(* Logix 5000 project; controller CarbonScout_MK6 vendor 1 type 14 code 154 rev 32.11; software revision 32.00; part 12 of 17 *)
(* tags used below, declared in another part *)
   DN_Cal : BOOL;   // Calculation Done Bit to proceed next step
   ExtraValvesAuto : BOOL;
   Index : DINT;
   InitialPurgeRequired : BOOL;
   LocalSampleTank : DINT;
   ONS : BOOL[32];
   TimeCompare : TimerCompare;
   AI_LIT_01 : P_AIn;   // Carbon Scout Laser Level Transmitter
   AI_LIT_02 : P_AIn;   // Carbon Scout Cone Level Transmitter
   AI_WIT_01 : P_AIn;   // Weight measure
   CS_Alarms : P_Alarm[80];
   CS_DINTParams : DINT[100];
   CS_REALParams : REAL[80];   // CS REAL Parameters
   CS_Result : CS_Results;   // Sample Result Live Async
   CS_ResultStore : CS_Results[20,20];   // Sample Result Historical
   CS_SampleSeq : DINT[129];
   CS_Seq : GEK_Sequence;
   CS_Seq_ControlStop : BOOL;
   CS_Tank : CS_TankParams[20];
   CS_TankOrder : DINT[17];
   CS_Timer : TIMER[80];
   CS_XRF : XRF;
   CS_XRF_DetTemp : REAL;   // Used in ewon for data records
   CS_XRF_ProbeTemp : REAL;
   FOQ01 : TOTALIZER;   // PurgeTotaliser
   N51 : DINT[5];   // From Client
   Oneshot2 : DINT;
   Oneshot3 : DINT;
   Simulation : DINT;
   TankPointer : DINT;
   TimeAndDate : DINT[7];
   Valve_SPR_01 : P_ValveSO;   // Air injection valve
   Valve_XV_01 : P_ValveSO;   // Sample Valve Tank 1
   Valve_XV_02 : P_ValveSO;   // Sample Valve Tank 2
   Valve_XV_03 : P_ValveSO;   // Sample Valve Tank 3
   Valve_XV_04 : P_ValveSO;   // Sample Valve Tank 4
   Valve_XV_05 : P_ValveSO;   // Sample Valve Tank 5
   Valve_XV_06 : P_ValveSO;   // Sample Valve Tank 6
   Valve_XV_07 : P_ValveSO;   // Sample Valve Tank 7
   Valve_XV_08 : P_ValveSO;   // Sample Valve Tank 8
   Valve_XV_09 : P_ValveSO;   // Sample Valve Tank 9
   Valve_XV_10 : P_ValveSO;   // Sample Valve Tank 10
   Valve_XV_11 : P_ValveSO;   // Purge Valve
   Valve_XV_12 : P_ValveSO;   // Slurry inlet vavle
   Valve_XV_13 : P_ValveSO;   // Sample line vavle
   Valve_XV_14 : P_ValveSO;   // Top wash vavle
   Valve_XV_15 : P_ValveSO;   // Bottme wash vavle
   Valve_XV_16 : P_ValveSO;   // Potable water valve / Supply Water Valve
   Valve_XV_17 : P_ValveSO;   // Sample cone outlet vavle
   Valve_XV_18 : P_ValveSO;   // Sample strainer discharge
   Valve_XV_19 : P_ValveSO;   // Laser window
   Valve_XV_21_30 : P_ValveSO;   // Sample isolation valve
   Valve_XV_30 : P_ValveSO;   // XRF cooling valve
   Valve_XV_40 : P_ValveSO;   // XRF power on valve
   XV2130ClosedOnce : BOOL;
(* SeqProgram, continued *)

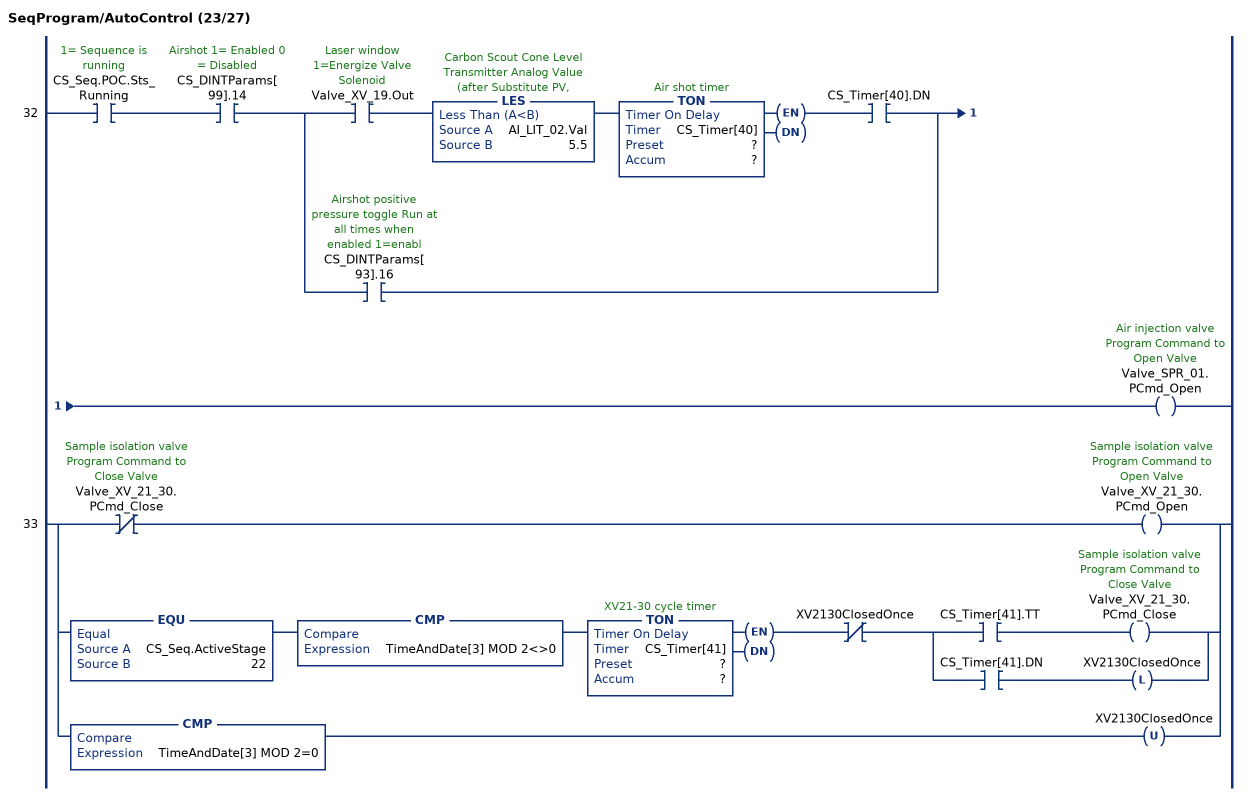
   [picture p234: SeqProgram/AutoControl rungs 32-33]
   32: XIC(CS_Seq.POC.Sts_Running)XIC(CS_DINTParams[99].14)[XIC(Valve_XV_19.Out) LES(AI_LIT_02.Val,5.5) TON(CS_Timer[40],?,?) XIC(CS_Timer[40].DN) ,XIC(CS_DINTParams[93].16) ]OTE(Valve_SPR_01.PCmd_Open);
   33: [XIO(Valve_XV_21_30.PCmd_Close) OTE(Valve_XV_21_30.PCmd_Open) ,EQU(CS_Seq.ActiveStage,22) CMP(TimeAndDate[3] MOD 2<>0) TON(CS_Timer[41],?,?) XIO(XV2130ClosedOnce) [XIC(CS_Timer[41].TT) OTE(Valve_XV_21_30.PCmd_Close) ,XIC(CS_Timer[41].DN) OTL(XV2130ClosedOnce) ] ,CMP(TimeAndDate[3] MOD 2=0) OTU(XV2130ClosedOnce) ];
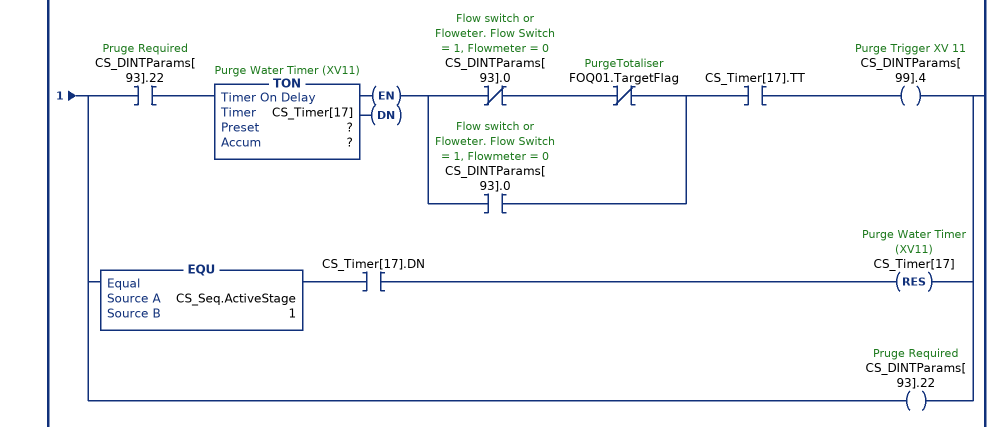
   // Purge Requests
   34: [[[[XIC(CS_DINTParams[99].28) ,XIC(InitialPurgeRequired) ] EQU(CS_Seq.ActiveStage,4) ,EQU(CS_Seq.ActiveStage,13) ] ,XIC(CS_DINTParams[99].4) ] XIC(CS_Seq.POC.Sts_Running) ,[EQU(CS_DINTParams[2],1) XIC(CS_Alarms[14].Alm) XIC(Valve_XV_12.Sts_Closed) ,EQU(CS_DINTParams[2],2) XIC(CS_Alarms[15].Alm) XIC(Valve_XV_12.Sts_Closed) ,EQU(CS_DINTParams[2],3) XIC(CS_Alarms[16].Alm) XIC(Valve_XV_12.Sts_Closed) ,EQU(CS_DINTParams[2],4) XIC(CS_Alarms[17].Alm) XIC(Valve_XV_12.Sts_Closed) ,EQU(CS_DINTParams[2],5) XIC(CS_Alarms[18].Alm) XIC(Valve_XV_12.Sts_Closed) ,EQU(CS_DINTParams[2],6) XIC(CS_Alarms[19].Alm) XIC(Valve_XV_12.Sts_Closed) ,EQU(CS_DINTParams[2],7) XIC(CS_Alarms[20].Alm) XIC(Valve_XV_12.Sts_Closed) ,EQU(CS_DINTParams[2],8) XIC(CS_Alarms[21].Alm) XIC(Valve_XV_12.Sts_Closed) ,EQU(CS_DINTParams[2],9) XIC(CS_Alarms[22].Alm) XIC(Valve_XV_12.Sts_Closed) ,EQU(CS_DINTParams[2],10) XIC(CS_Alarms[23].Alm) XIC(Valve_XV_12.Sts_Closed) ,XIC(CS_DINTParams[99].18) [EQU(CS_DINTParams[2],11) XIC(CS_Alarms[57].Alm) XIC(Valve_XV_12.Sts_Closed) ,EQU(CS_DINTParams[2],12) XIC(CS_Alarms[58].Alm) XIC(Valve_XV_12.Sts_Closed) ,EQU(CS_DINTParams[2],13) XIC(CS_Alarms[59].Alm) XIC(Valve_XV_12.Sts_Closed) ,EQU(CS_DINTParams[2],14) XIC(CS_Alarms[60].Alm) XIC(Valve_XV_12.Sts_Closed) ,EQU(CS_DINTParams[2],15) XIC(CS_Alarms[61].Alm) XIC(Valve_XV_12.Sts_Closed) ,EQU(CS_DINTParams[2],16) XIC(CS_Alarms[62].Alm) XIC(Valve_XV_12.Sts_Closed) ] ] XIO(CS_Seq.POC.Sts_Running) ][XIC(CS_DINTParams[93].22) TON(CS_Timer[17],?,?) [XIO(CS_DINTParams[93].0) XIO(FOQ01.TargetFlag) ,XIC(CS_DINTParams[93].0) ] XIC(CS_Timer[17].TT) OTE(CS_DINTParams[99].4) ,EQU(CS_Seq.ActiveStage,1) XIC(CS_Timer[17].DN) RES(CS_Timer[17]) ,OTE(CS_DINTParams[93].22) ];
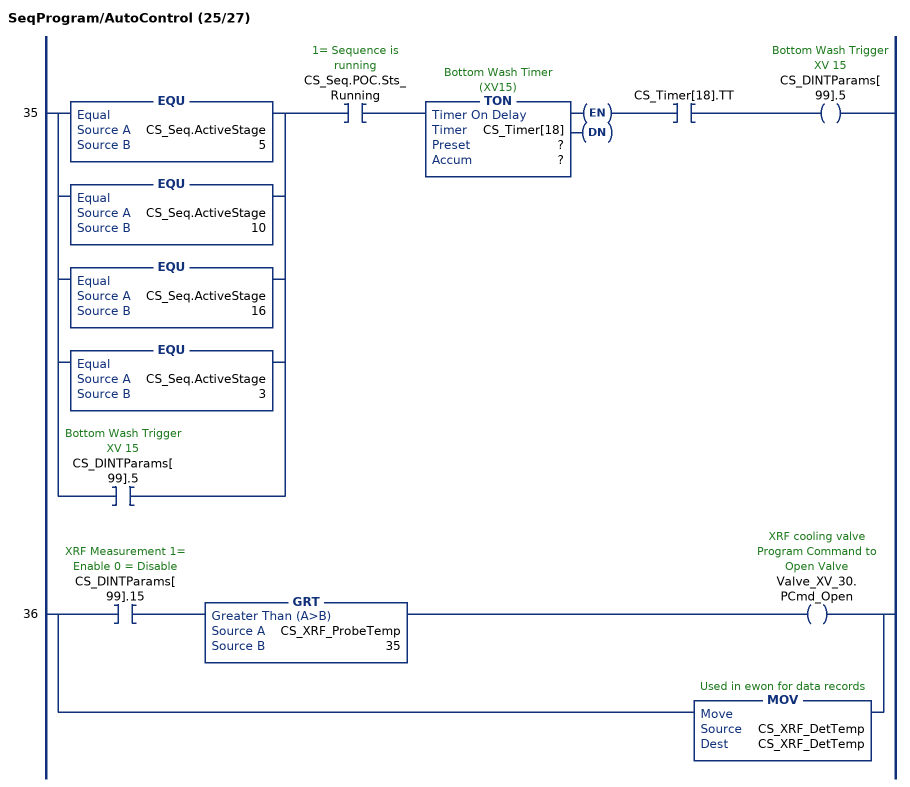
   35: [[EQU(CS_Seq.ActiveStage,5) ,EQU(CS_Seq.ActiveStage,10) ,EQU(CS_Seq.ActiveStage,16) ,EQU(CS_Seq.ActiveStage,3) ] ,XIC(CS_DINTParams[99].5) ]XIC(CS_Seq.POC.Sts_Running)TON(CS_Timer[18],?,?)XIC(CS_Timer[18].TT)OTE(CS_DINTParams[99].5);
   36: [XIC(CS_DINTParams[99].15) GRT(CS_XRF_ProbeTemp,35) OTE(Valve_XV_30.PCmd_Open) ,MOV(CS_XRF_DetTemp,CS_XRF_DetTemp) ];
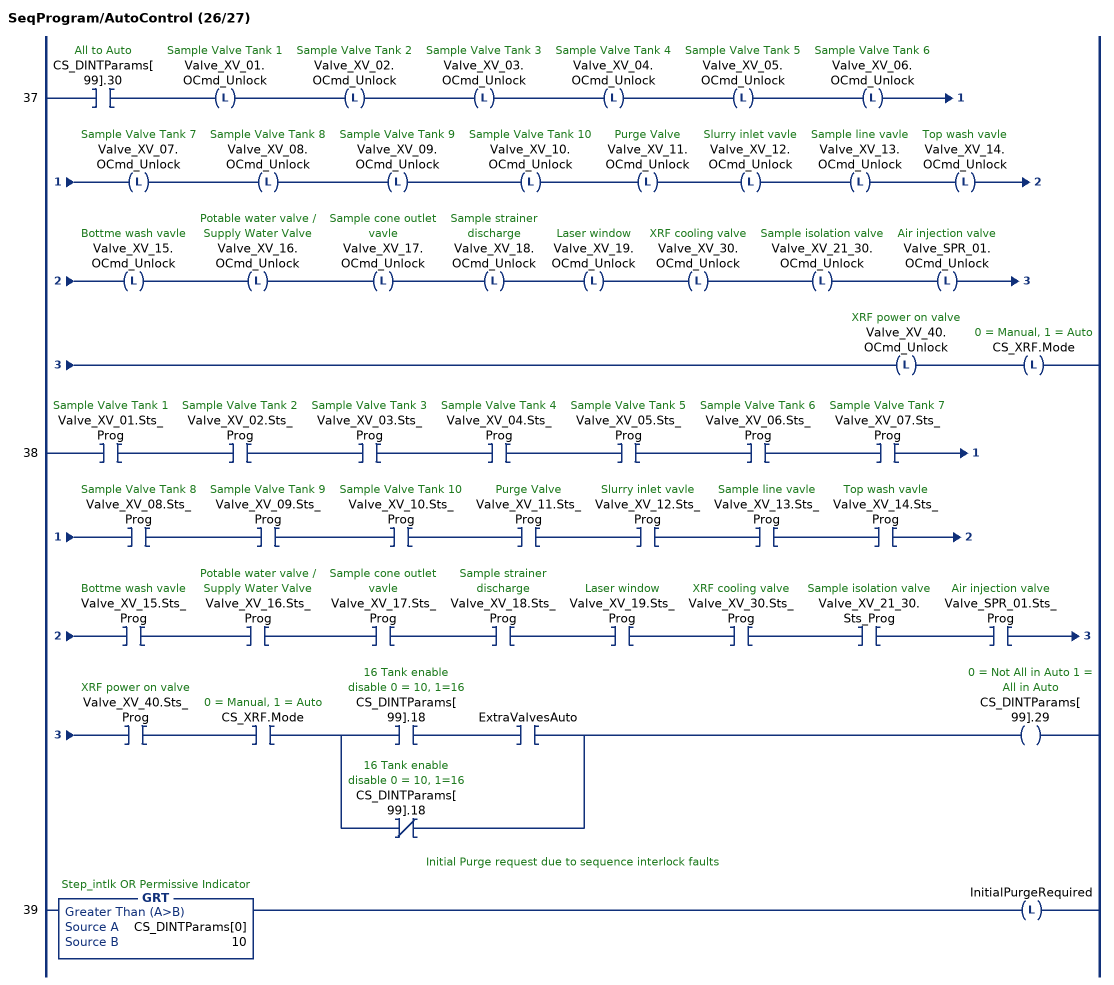
   37: XIC(CS_DINTParams[99].30)OTL(Valve_XV_01.OCmd_Unlock)OTL(Valve_XV_02.OCmd_Unlock)OTL(Valve_XV_03.OCmd_Unlock)OTL(Valve_XV_04.OCmd_Unlock)OTL(Valve_XV_05.OCmd_Unlock)OTL(Valve_XV_06.OCmd_Unlock)OTL(Valve_XV_07.OCmd_Unlock)OTL(Valve_XV_08.OCmd_Unlock)OTL(Valve_XV_09.OCmd_Unlock)OTL(Valve_XV_10.OCmd_Unlock)OTL(Valve_XV_11.OCmd_Unlock)OTL(Valve_XV_12.OCmd_Unlock)OTL(Valve_XV_13.OCmd_Unlock)OTL(Valve_XV_14.OCmd_Unlock)OTL(Valve_XV_15.OCmd_Unlock)OTL(Valve_XV_16.OCmd_Unlock)OTL(Valve_XV_17.OCmd_Unlock)OTL(Valve_XV_18.OCmd_Unlock)OTL(Valve_XV_19.OCmd_Unlock)OTL(Valve_XV_30.OCmd_Unlock)OTL(Valve_XV_21_30.OCmd_Unlock)OTL(Valve_SPR_01.OCmd_Unlock)OTL(Valve_XV_40.OCmd_Unlock)OTL(CS_XRF.Mode);
   38: XIC(Valve_XV_01.Sts_Prog)XIC(Valve_XV_02.Sts_Prog)XIC(Valve_XV_03.Sts_Prog)XIC(Valve_XV_04.Sts_Prog)XIC(Valve_XV_05.Sts_Prog)XIC(Valve_XV_06.Sts_Prog)XIC(Valve_XV_07.Sts_Prog)XIC(Valve_XV_08.Sts_Prog)XIC(Valve_XV_09.Sts_Prog)XIC(Valve_XV_10.Sts_Prog)XIC(Valve_XV_11.Sts_Prog)XIC(Valve_XV_12.Sts_Prog)XIC(Valve_XV_13.Sts_Prog)XIC(Valve_XV_14.Sts_Prog)XIC(Valve_XV_15.Sts_Prog)XIC(Valve_XV_16.Sts_Prog)XIC(Valve_XV_17.Sts_Prog)XIC(Valve_XV_18.Sts_Prog)XIC(Valve_XV_19.Sts_Prog)XIC(Valve_XV_30.Sts_Prog)XIC(Valve_XV_21_30.Sts_Prog)XIC(Valve_SPR_01.Sts_Prog)XIC(Valve_XV_40.Sts_Prog)XIC(CS_XRF.Mode)[XIC(CS_DINTParams[99].18) XIC(ExtraValvesAuto) ,XIO(CS_DINTParams[99].18) ]OTE(CS_DINTParams[99].29);
   // Initial Purge request due to sequence interlock faults
   39: GRT(CS_DINTParams[0],10)OTL(InitialPurgeRequired);
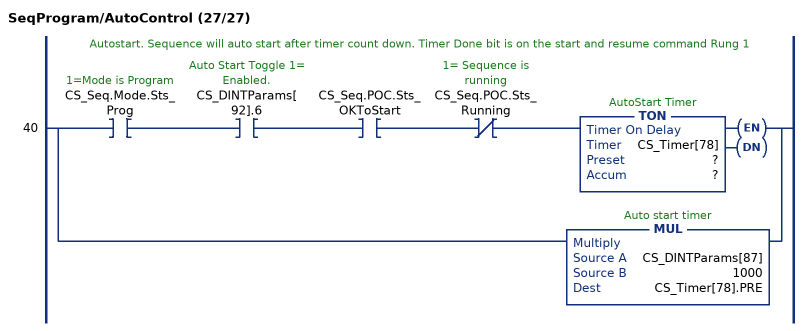
   // Autostart. Sequence will auto start after timer count down. Timer Done bit is on the start and resume command Rung 1
   40: [XIC(CS_Seq.Mode.Sts_Prog) XIC(CS_DINTParams[92].6) XIC(CS_Seq.POC.Sts_OKToStart) XIO(CS_Seq.POC.Sts_Running) TON(CS_Timer[78],?,?) ,MUL(CS_DINTParams[87],1000,CS_Timer[78].PRE) ];
END_ROUTINE

ROUTINE AutoTransition   (* ladder *)
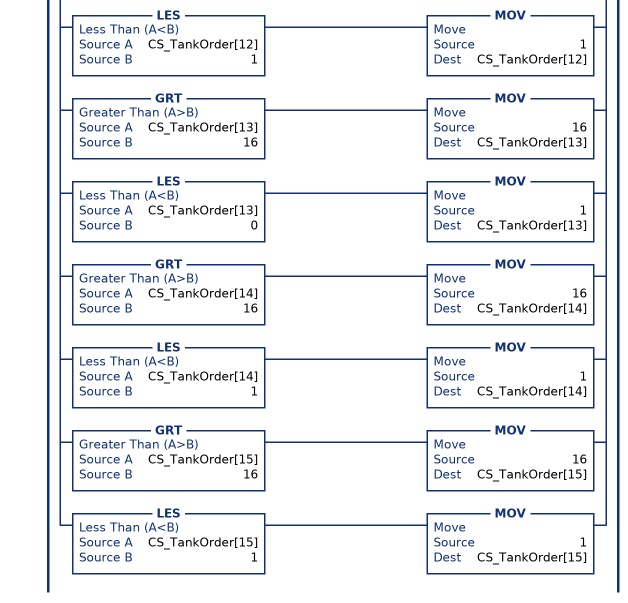
   // Tank order capping
   0: [GRT(CS_TankOrder[0],16) MOV(16,CS_TankOrder[0]) ,LES(CS_TankOrder[0],1) MOV(1,CS_TankOrder[0]) ,GRT(CS_TankOrder[1],16) MOV(16,CS_TankOrder[1]) ,LES(CS_TankOrder[1],1) MOV(1,CS_TankOrder[1]) ,GRT(CS_TankOrder[2],16) MOV(16,CS_TankOrder[2]) ,LES(CS_TankOrder[2],1) MOV(1,CS_TankOrder[2]) ,GRT(CS_TankOrder[3],16) MOV(16,CS_TankOrder[3]) ,LES(CS_TankOrder[3],1) MOV(1,CS_TankOrder[3]) ,GRT(CS_TankOrder[4],16) MOV(16,CS_TankOrder[4]) ,LES(CS_TankOrder[4],1) MOV(1,CS_TankOrder[4]) ,GRT(CS_TankOrder[5],16) MOV(16,CS_TankOrder[5]) ,LES(CS_TankOrder[5],1) MOV(1,CS_TankOrder[5]) ,GRT(CS_TankOrder[6],16) MOV(16,CS_TankOrder[6]) ,LES(CS_TankOrder[6],1) MOV(1,CS_TankOrder[6]) ,GRT(CS_TankOrder[7],16) MOV(16,CS_TankOrder[7]) ,LES(CS_TankOrder[7],1) MOV(1,CS_TankOrder[7]) ,GRT(CS_TankOrder[8],16) MOV(16,CS_TankOrder[8]) ,LES(CS_TankOrder[8],1) MOV(1,CS_TankOrder[8]) ,GRT(CS_TankOrder[9],16) MOV(16,CS_TankOrder[9]) ,LES(CS_TankOrder[9],1) MOV(1,CS_TankOrder[9]) ,GRT(CS_TankOrder[10],16) MOV(16,CS_TankOrder[10]) ,LES(CS_TankOrder[10],1) MOV(1,CS_TankOrder[10]) ,GRT(CS_TankOrder[11],16) MOV(16,CS_TankOrder[11]) ,LES(CS_TankOrder[11],1) MOV(1,CS_TankOrder[11]) ,GRT(CS_TankOrder[12],16) MOV(16,CS_TankOrder[12]) ,LES(CS_TankOrder[12],1) MOV(1,CS_TankOrder[12]) ,GRT(CS_TankOrder[13],16) MOV(16,CS_TankOrder[13]) ,LES(CS_TankOrder[13],0) MOV(1,CS_TankOrder[13]) ,GRT(CS_TankOrder[14],16) MOV(16,CS_TankOrder[14]) ,LES(CS_TankOrder[14],1) MOV(1,CS_TankOrder[14]) ,GRT(CS_TankOrder[15],16) MOV(16,CS_TankOrder[15]) ,LES(CS_TankOrder[15],1) MOV(1,CS_TankOrder[15]) ];
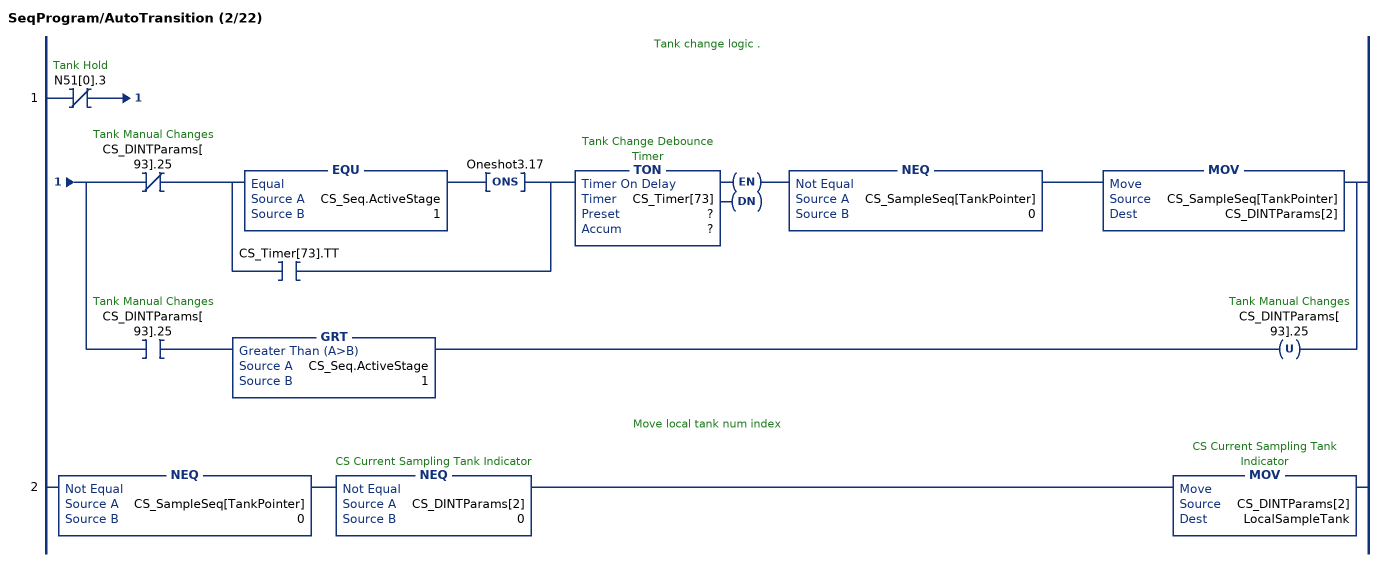
   // Tank change logic .
   1: XIO(N51[0].3)[XIO(CS_DINTParams[93].25) [EQU(CS_Seq.ActiveStage,1) ONS(Oneshot3.17) ,XIC(CS_Timer[73].TT) ] TON(CS_Timer[73],?,?) NEQ(CS_SampleSeq[TankPointer],0) MOV(CS_SampleSeq[TankPointer],CS_DINTParams[2]) ,XIC(CS_DINTParams[93].25) GRT(CS_Seq.ActiveStage,1) OTU(CS_DINTParams[93].25) ];
   // Move local tank num index
   2: NEQ(CS_SampleSeq[TankPointer],0)NEQ(CS_DINTParams[2],0)MOV(CS_DINTParams[2],LocalSampleTank);
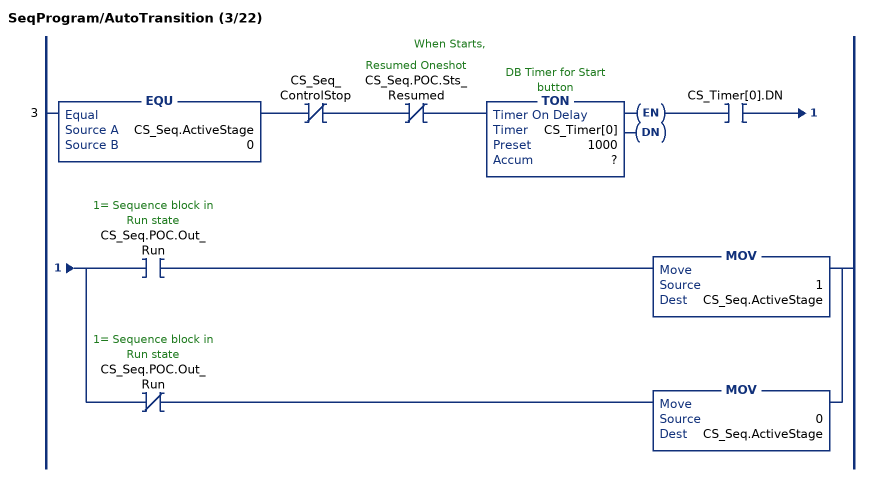
   // When Starts,
   3: EQU(CS_Seq.ActiveStage,0)XIO(CS_Seq_ControlStop)XIO(CS_Seq.POC.Sts_Resumed)TON(CS_Timer[0],?,?)XIC(CS_Timer[0].DN)[XIC(CS_Seq.POC.Out_Run) MOV(1,CS_Seq.ActiveStage) ,XIO(CS_Seq.POC.Out_Run) MOV(0,CS_Seq.ActiveStage) ];
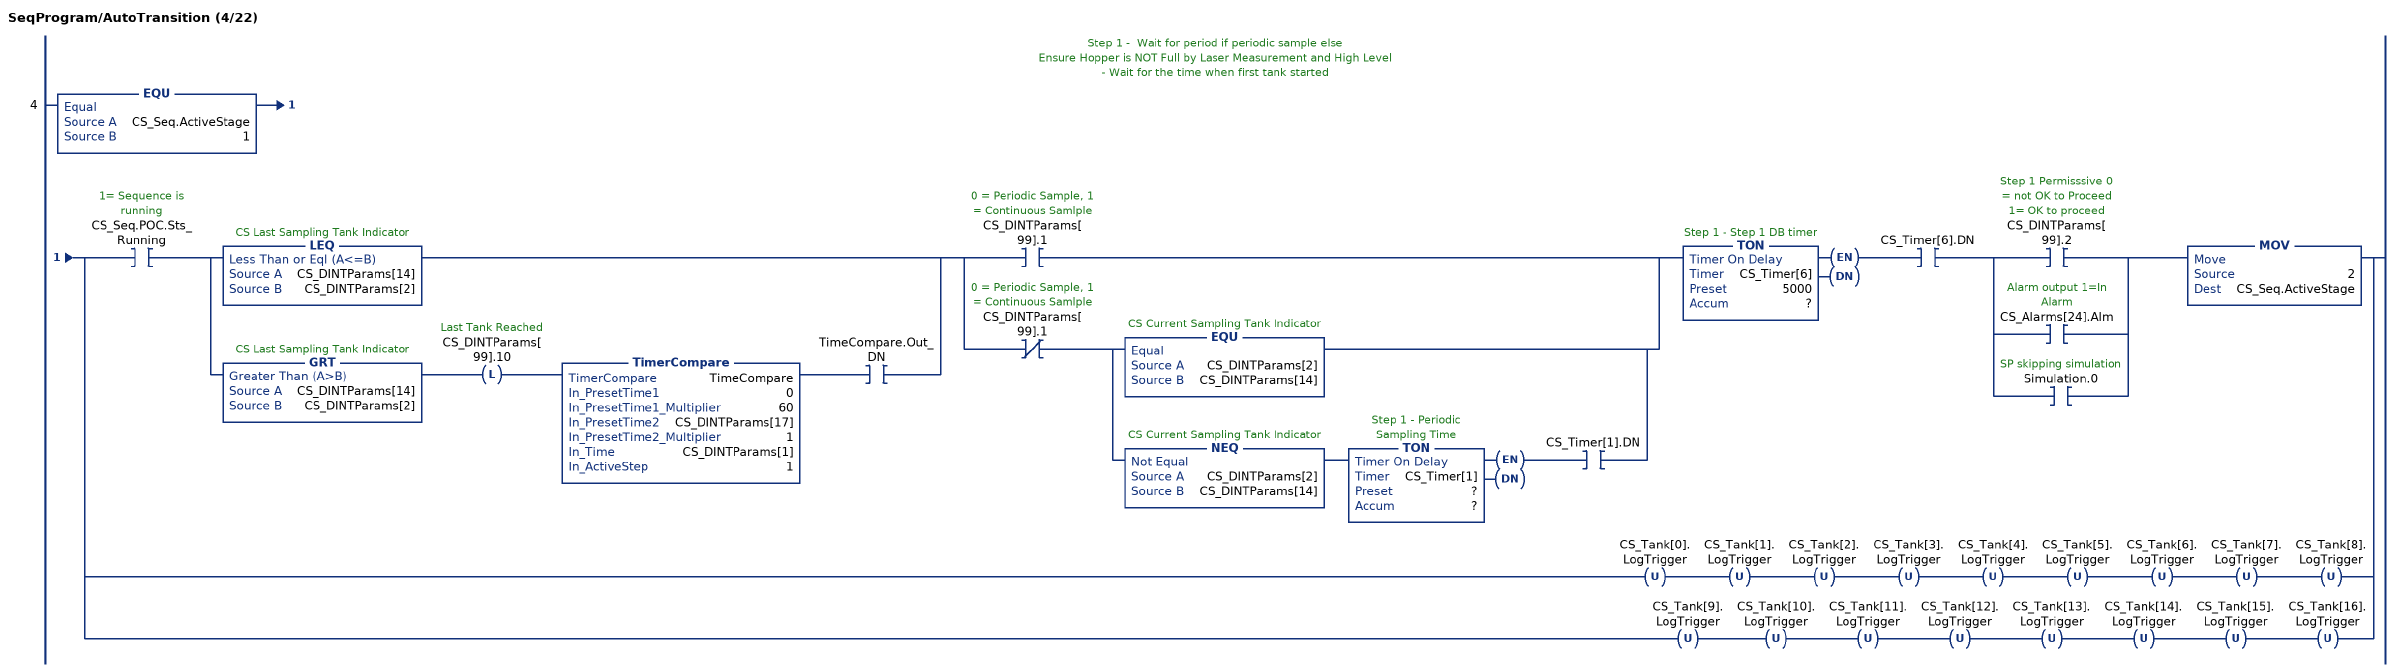
   // Step 1 -  Wait for period if periodic sample else
   // Ensure Hopper is NOT Full by Laser Measurement and High Level
   // - Wait for the time when first tank started
   4: EQU(CS_Seq.ActiveStage,1)[XIC(CS_Seq.POC.Sts_Running) [LEQ(CS_DINTParams[14],CS_DINTParams[2]) ,GRT(CS_DINTParams[14],CS_DINTParams[2]) OTL(CS_DINTParams[99].10) TimerCompare(TimeCompare,0,60,CS_DINTParams[17],1,CS_DINTParams[1],1) XIC(TimeCompare.Out_DN) ] [XIC(CS_DINTParams[99].1) ,XIO(CS_DINTParams[99].1) [EQU(CS_DINTParams[2],CS_DINTParams[14]) ,NEQ(CS_DINTParams[2],CS_DINTParams[14]) TON(CS_Timer[1],?,?) XIC(CS_Timer[1].DN) ] ] TON(CS_Timer[6],?,?) XIC(CS_Timer[6].DN) [[XIC(CS_DINTParams[99].2) ,XIC(CS_Alarms[24].Alm) ] ,XIC(Simulation.0) ] MOV(2,CS_Seq.ActiveStage) ,OTU(CS_Tank[0].LogTrigger) OTU(CS_Tank[1].LogTrigger) OTU(CS_Tank[2].LogTrigger) OTU(CS_Tank[3].LogTrigger) OTU(CS_Tank[4].LogTrigger) OTU(CS_Tank[5].LogTrigger) OTU(CS_Tank[6].LogTrigger) OTU(CS_Tank[7].LogTrigger) OTU(CS_Tank[8].LogTrigger) ,OTU(CS_Tank[9].LogTrigger) OTU(CS_Tank[10].LogTrigger) OTU(CS_Tank[11].LogTrigger) OTU(CS_Tank[12].LogTrigger) OTU(CS_Tank[13].LogTrigger) OTU(CS_Tank[14].LogTrigger) OTU(CS_Tank[15].LogTrigger) OTU(CS_Tank[16].LogTrigger) ];
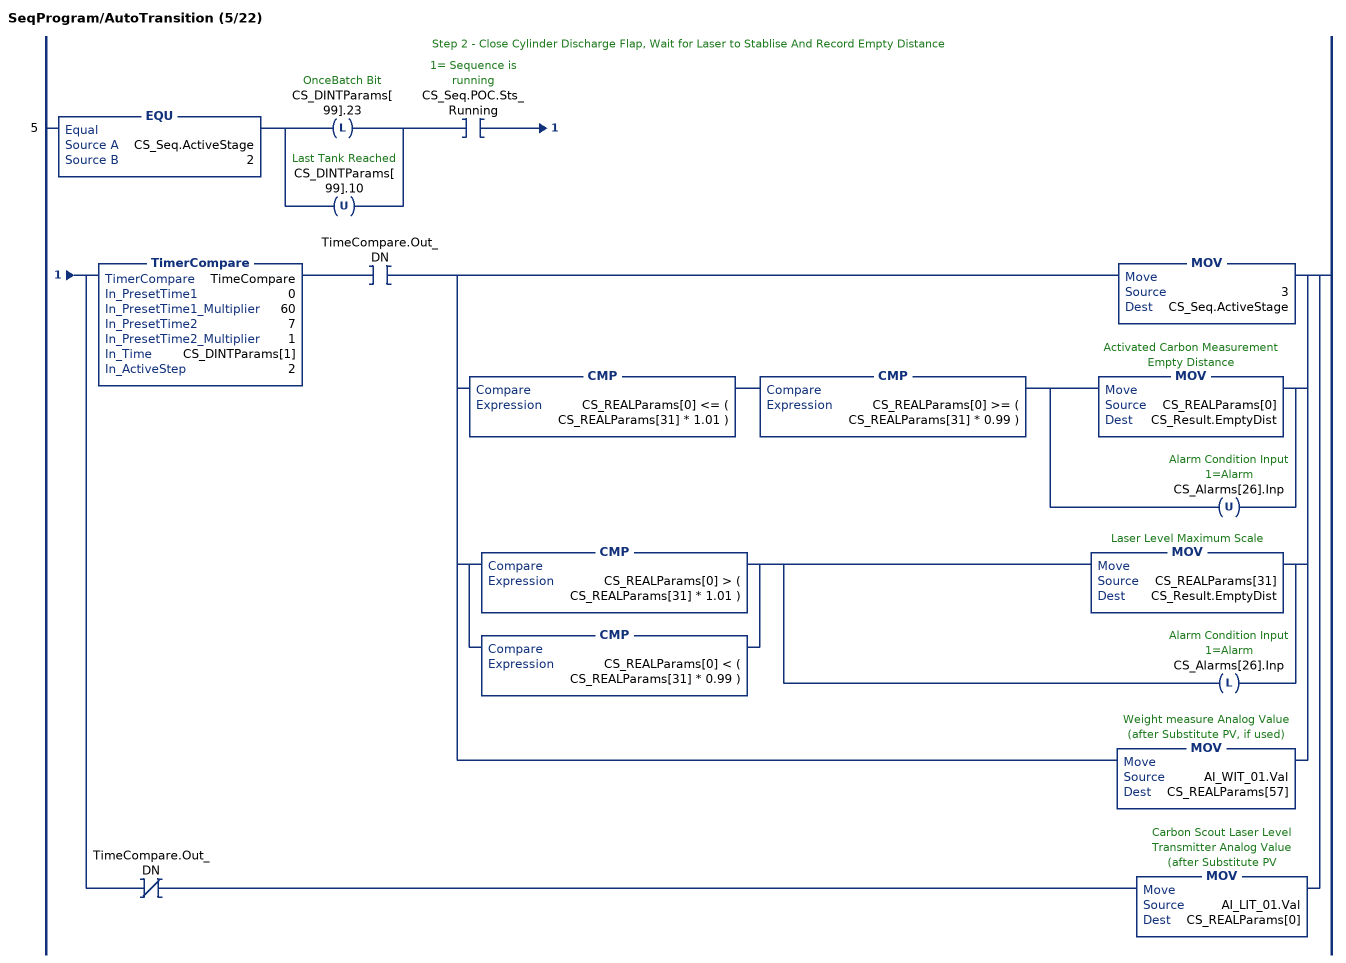
   // Step 2 - Close Cylinder Discharge Flap, Wait for Laser to Stablise And Record Empty Distance
   5: EQU(CS_Seq.ActiveStage,2)[OTL(CS_DINTParams[99].23) ,OTU(CS_DINTParams[99].10) ]XIC(CS_Seq.POC.Sts_Running)[TimerCompare(TimeCompare,0,60,7,1,CS_DINTParams[1],2) XIC(TimeCompare.Out_DN) [MOV(3,CS_Seq.ActiveStage) ,[CMP(CS_REALParams[0] <= ( CS_REALParams[31] * 1.01 )) CMP(CS_REALParams[0] >= ( CS_REALParams[31] * 0.99 )) [MOV(CS_REALParams[0],CS_Result.EmptyDist) ,OTU(CS_Alarms[26].Inp) ] ,[CMP(CS_REALParams[0] > ( CS_REALParams[31] * 1.01 )) ,CMP(CS_REALParams[0] < ( CS_REALParams[31] * 0.99 )) ] [MOV(CS_REALParams[31],CS_Result.EmptyDist) ,OTL(CS_Alarms[26].Inp) ] ,MOV(AI_WIT_01.Val,CS_REALParams[57]) ] ] ,XIO(TimeCompare.Out_DN) MOV(AI_LIT_01.Val,CS_REALParams[0]) ];
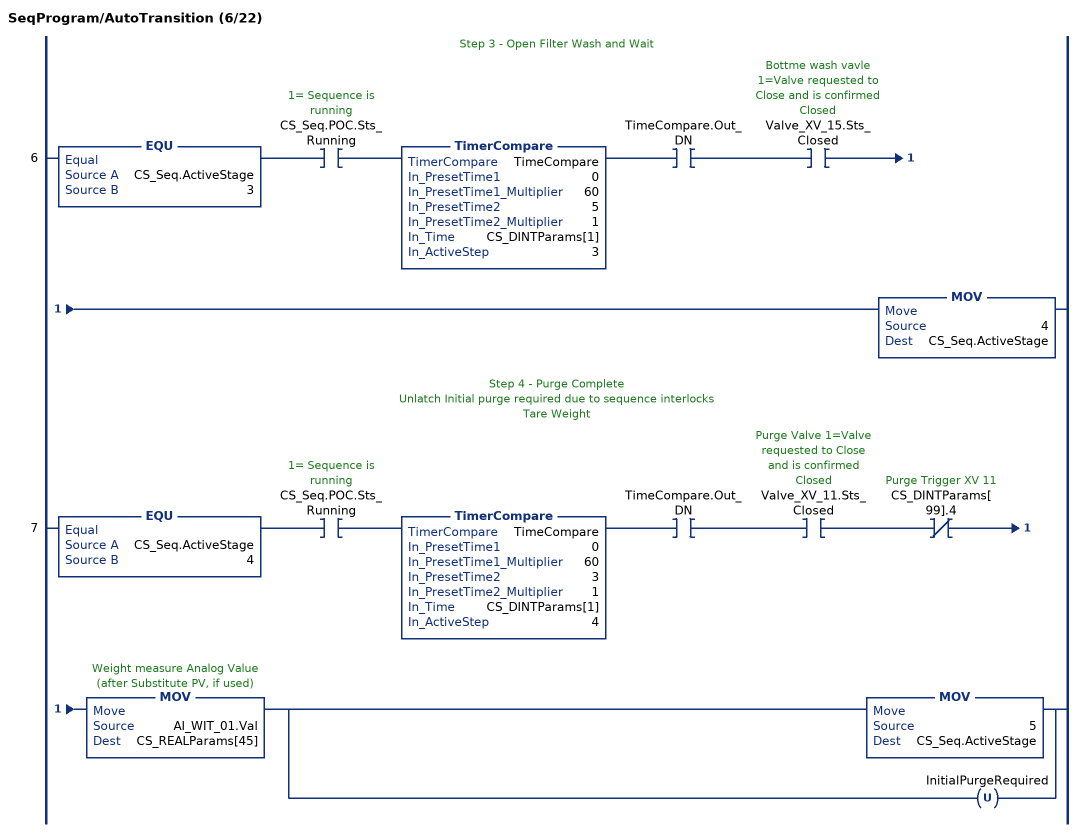
   // Step 3 - Open Filter Wash and Wait
   6: EQU(CS_Seq.ActiveStage,3)XIC(CS_Seq.POC.Sts_Running)TimerCompare(TimeCompare,0,60,5,1,CS_DINTParams[1],3)XIC(TimeCompare.Out_DN)XIC(Valve_XV_15.Sts_Closed)MOV(4,CS_Seq.ActiveStage);
   // Step 4 - Purge Complete
   // Unlatch Initial purge required due to sequence interlocks
   // Tare Weight
   7: EQU(CS_Seq.ActiveStage,4)XIC(CS_Seq.POC.Sts_Running)TimerCompare(TimeCompare,0,60,3,1,CS_DINTParams[1],4)XIC(TimeCompare.Out_DN)XIC(Valve_XV_11.Sts_Closed)XIO(CS_DINTParams[99].4)MOV(AI_WIT_01.Val,CS_REALParams[45])[MOV(5,CS_Seq.ActiveStage) ,OTU(InitialPurgeRequired) ];
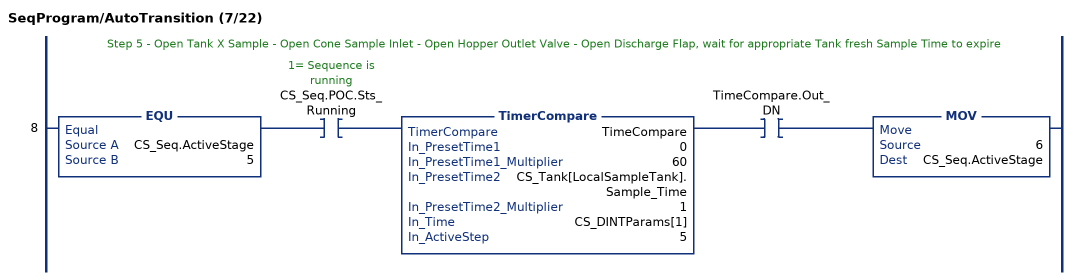
   // Step 5 - Open Tank X Sample - Open Cone Sample Inlet - Open Hopper Outlet Valve - Open Discharge Flap, wait for appropriate Tank fresh Sample Time to expire
   8: EQU(CS_Seq.ActiveStage,5)XIC(CS_Seq.POC.Sts_Running)TimerCompare(TimeCompare,0,60,CS_Tank[LocalSampleTank].Sample_Time,1,CS_DINTParams[1],5)XIC(TimeCompare.Out_DN)MOV(6,CS_Seq.ActiveStage);
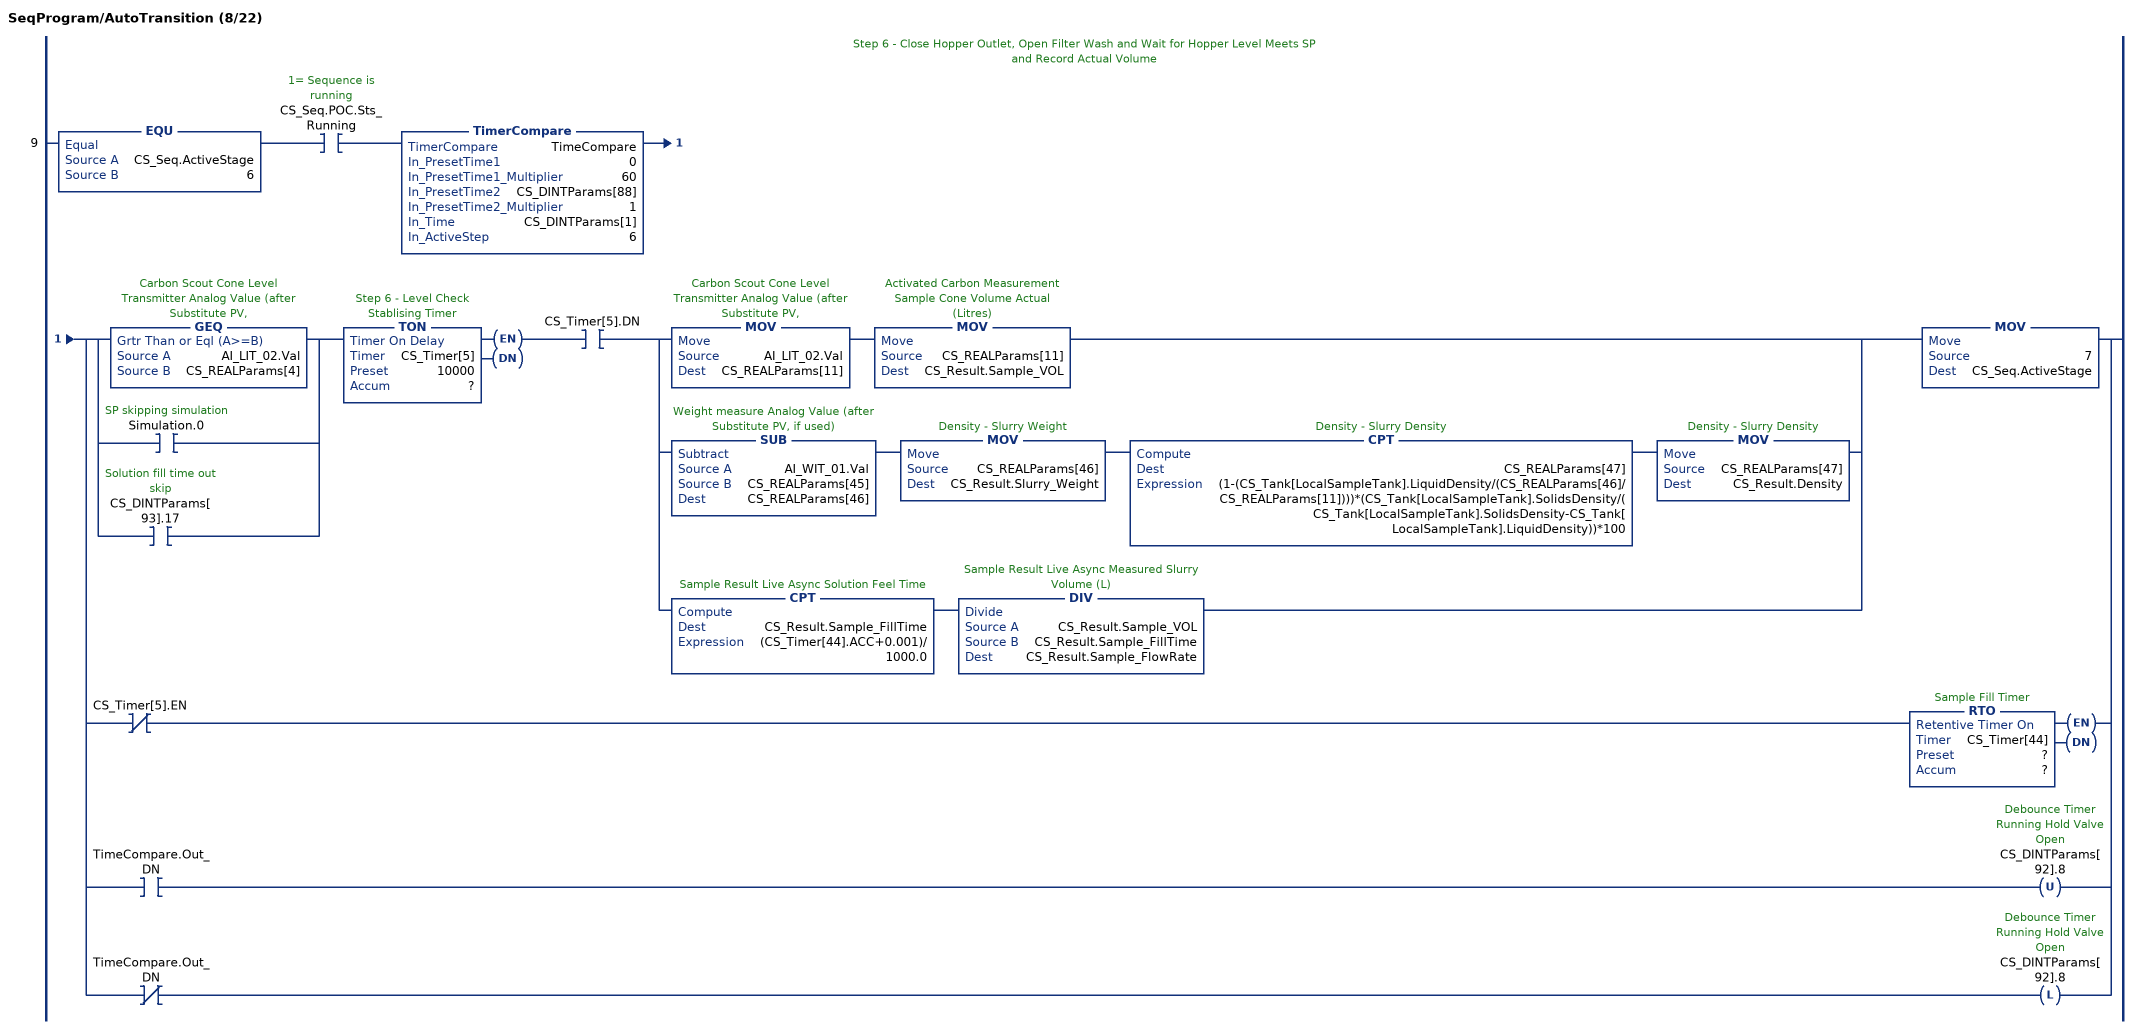
   // Step 6 - Close Hopper Outlet, Open Filter Wash and Wait for Hopper Level Meets SP
   // and Record Actual Volume
   9: EQU(CS_Seq.ActiveStage,6)XIC(CS_Seq.POC.Sts_Running)TimerCompare(TimeCompare,0,60,CS_DINTParams[88],1,CS_DINTParams[1],6)[[[GEQ(AI_LIT_02.Val,CS_REALParams[4]) ,XIC(Simulation.0) ,XIC(CS_DINTParams[93].17) ] TON(CS_Timer[5],?,?) XIC(CS_Timer[5].DN) [MOV(AI_LIT_02.Val,CS_REALParams[11]) MOV(CS_REALParams[11],CS_Result.Sample_VOL) ,SUB(AI_WIT_01.Val,CS_REALParams[45],CS_REALParams[46]) MOV(CS_REALParams[46],CS_Result.Slurry_Weight) CPT(CS_REALParams[47],(1-(CS_Tank[LocalSampleTank].LiquidDensity/(CS_REALParams[46]/CS_REALParams[11])))*(CS_Tank[LocalSampleTank].SolidsDensity/(CS_Tank[LocalSampleTank].SolidsDensity-CS_Tank[LocalSampleTank].LiquidDensity))*100) MOV(CS_REALParams[47],CS_Result.Density) ,CPT(CS_Result.Sample_FillTime,(CS_Timer[44].ACC+0.001)/1000.0) DIV(CS_Result.Sample_VOL,CS_Result.Sample_FillTime,CS_Result.Sample_FlowRate) ] MOV(7,CS_Seq.ActiveStage) ,XIO(CS_Timer[5].EN) RTO(CS_Timer[44],?,?) ] ,XIC(TimeCompare.Out_DN) OTU(CS_DINTParams[92].8) ,XIO(TimeCompare.Out_DN) OTL(CS_DINTParams[92].8) ];
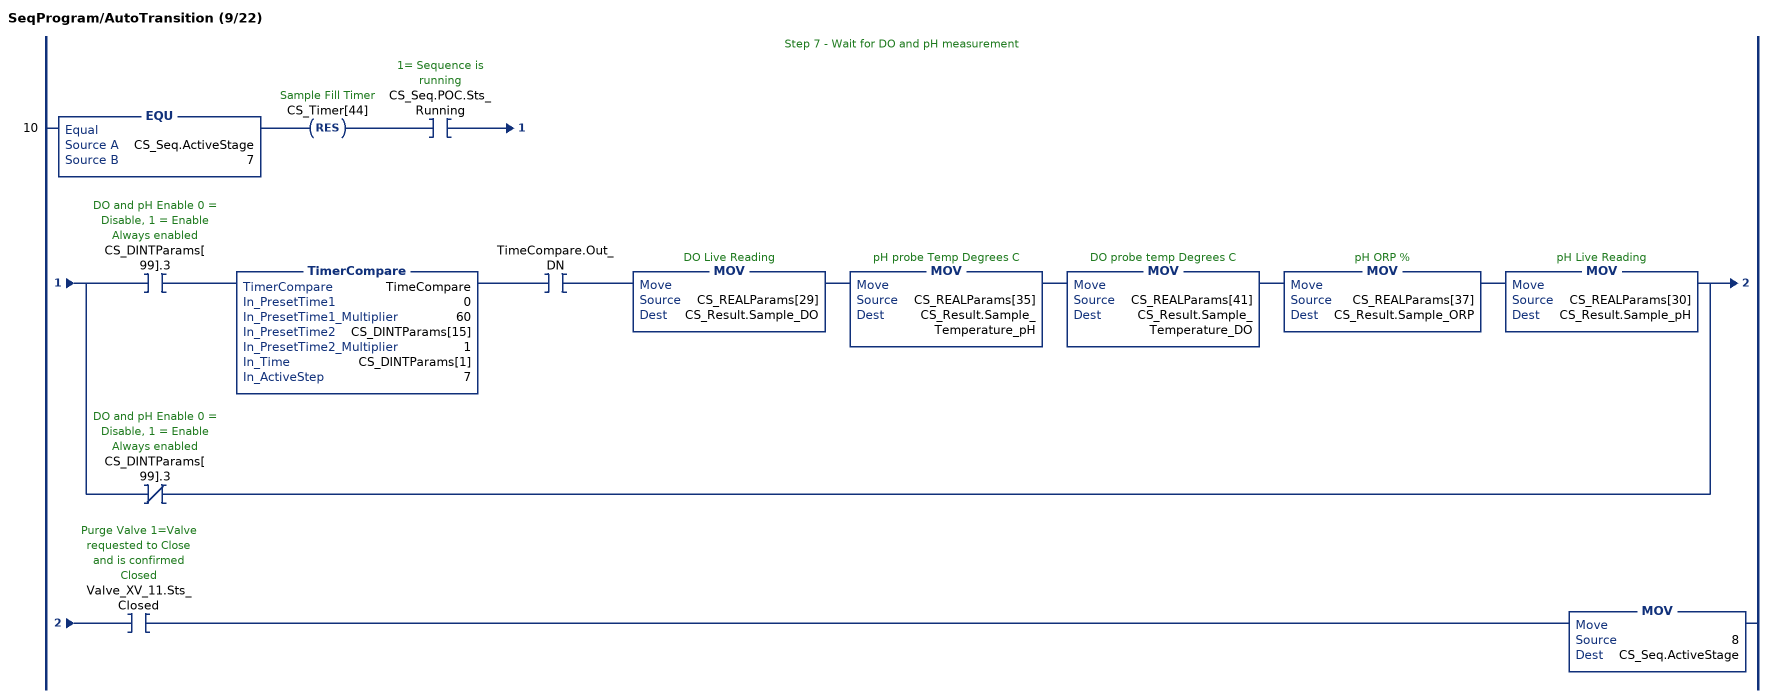
   // Step 7 - Wait for DO and pH measurement
   10: EQU(CS_Seq.ActiveStage,7)RES(CS_Timer[44])XIC(CS_Seq.POC.Sts_Running)[XIC(CS_DINTParams[99].3) TimerCompare(TimeCompare,0,60,CS_DINTParams[15],1,CS_DINTParams[1],7) XIC(TimeCompare.Out_DN) MOV(CS_REALParams[29],CS_Result.Sample_DO) MOV(CS_REALParams[35],CS_Result.Sample_Temperature_pH) MOV(CS_REALParams[41],CS_Result.Sample_Temperature_DO) MOV(CS_REALParams[37],CS_Result.Sample_ORP) MOV(CS_REALParams[30],CS_Result.Sample_pH) ,XIO(CS_DINTParams[99].3) ]XIC(Valve_XV_11.Sts_Closed)MOV(8,CS_Seq.ActiveStage);
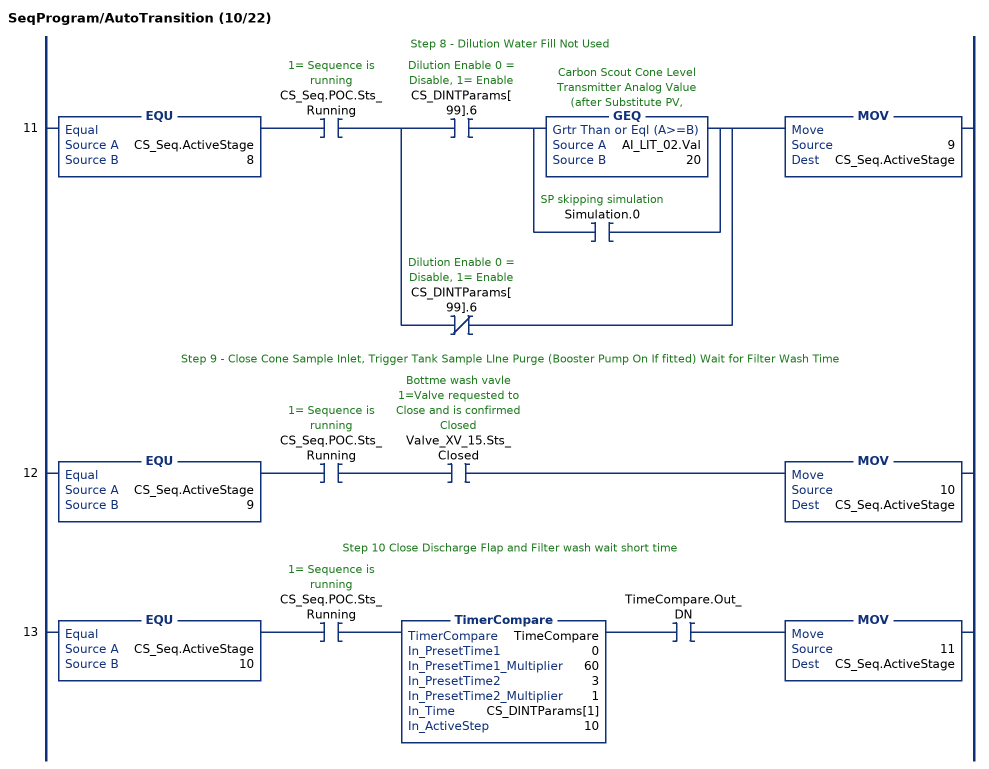
   // Step 8 - Dilution Water Fill Not Used
   11: EQU(CS_Seq.ActiveStage,8)XIC(CS_Seq.POC.Sts_Running)[XIC(CS_DINTParams[99].6) [GEQ(AI_LIT_02.Val,20) ,XIC(Simulation.0) ] ,XIO(CS_DINTParams[99].6) ]MOV(9,CS_Seq.ActiveStage);
   // Step 9 - Close Cone Sample Inlet, Trigger Tank Sample LIne Purge (Booster Pump On If fitted) Wait for Filter Wash Time
   12: EQU(CS_Seq.ActiveStage,9)XIC(CS_Seq.POC.Sts_Running)XIC(Valve_XV_15.Sts_Closed)MOV(10,CS_Seq.ActiveStage);
   // Step 10 Close Discharge Flap and Filter wash wait short time
   13: EQU(CS_Seq.ActiveStage,10)XIC(CS_Seq.POC.Sts_Running)TimerCompare(TimeCompare,0,60,3,1,CS_DINTParams[1],10)XIC(TimeCompare.Out_DN)MOV(11,CS_Seq.ActiveStage);
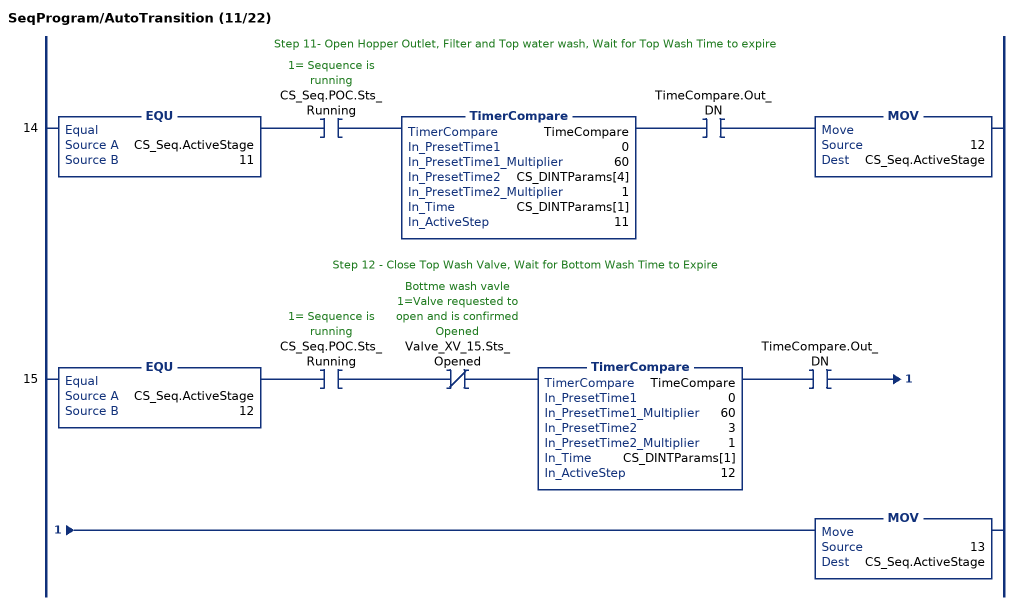
   // Step 11- Open Hopper Outlet, Filter and Top water wash, Wait for Top Wash Time to expire
   14: EQU(CS_Seq.ActiveStage,11)XIC(CS_Seq.POC.Sts_Running)TimerCompare(TimeCompare,0,60,CS_DINTParams[4],1,CS_DINTParams[1],11)XIC(TimeCompare.Out_DN)MOV(12,CS_Seq.ActiveStage);
   // Step 12 - Close Top Wash Valve, Wait for Bottom Wash Time to Expire
   15: EQU(CS_Seq.ActiveStage,12)XIC(CS_Seq.POC.Sts_Running)XIO(Valve_XV_15.Sts_Opened)TimerCompare(TimeCompare,0,60,3,1,CS_DINTParams[1],12)XIC(TimeCompare.Out_DN)MOV(13,CS_Seq.ActiveStage);
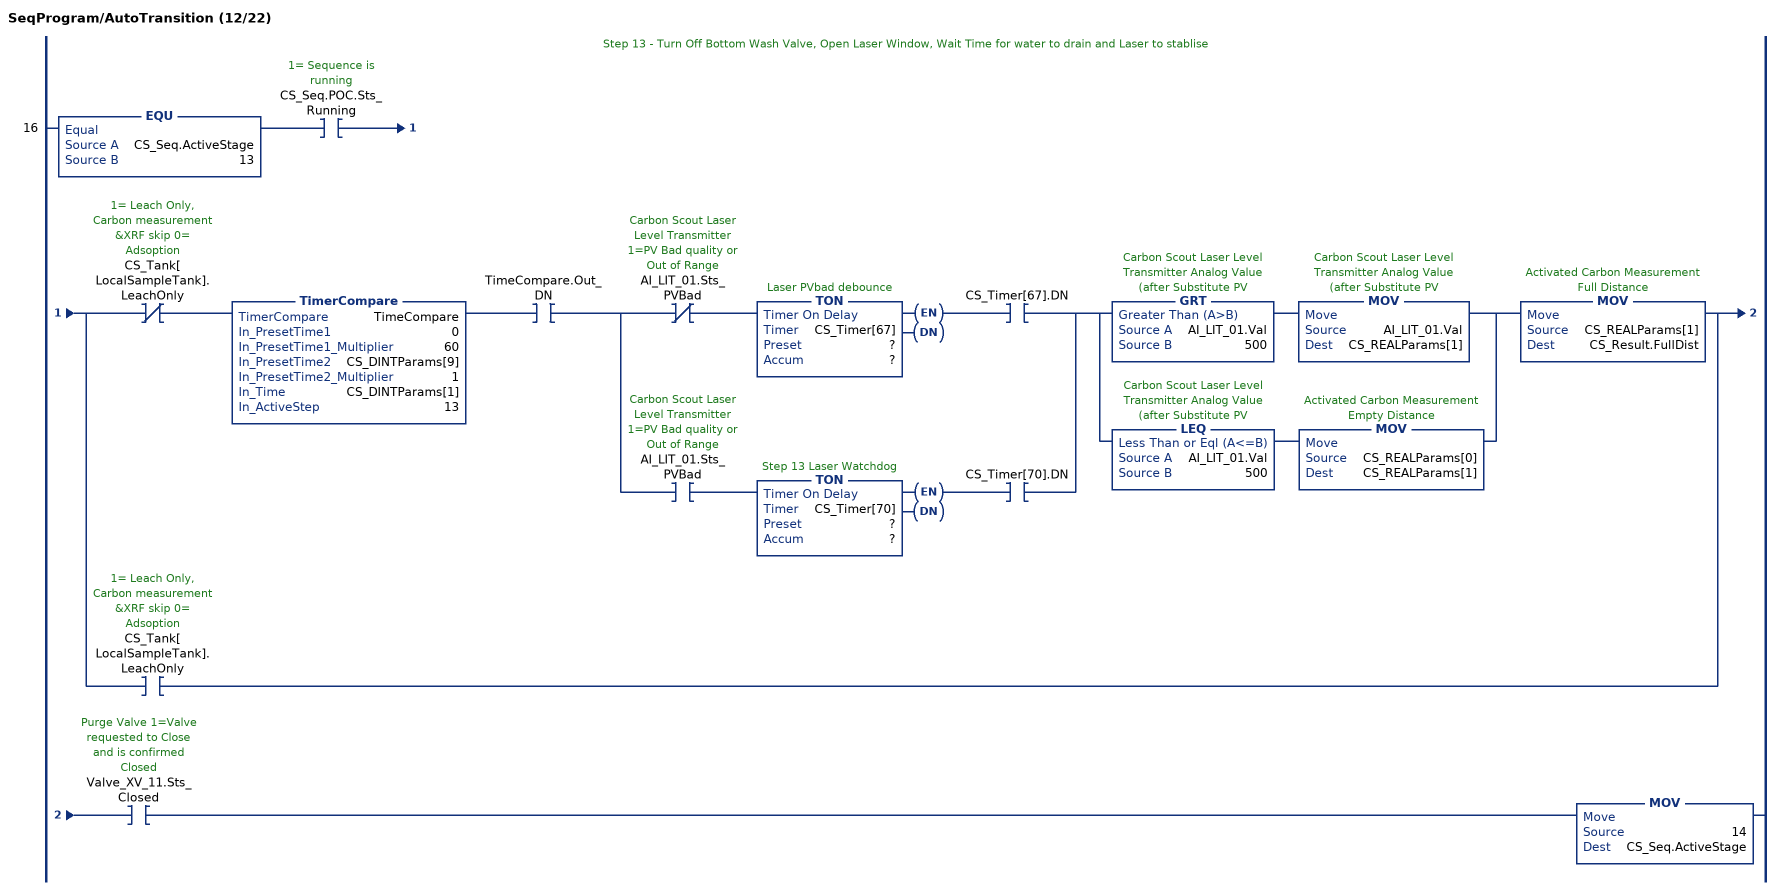
   // Step 13 - Turn Off Bottom Wash Valve, Open Laser Window, Wait Time for water to drain and Laser to stablise
   16: EQU(CS_Seq.ActiveStage,13)XIC(CS_Seq.POC.Sts_Running)[XIO(CS_Tank[LocalSampleTank].LeachOnly) TimerCompare(TimeCompare,0,60,CS_DINTParams[9],1,CS_DINTParams[1],13) XIC(TimeCompare.Out_DN) [XIO(AI_LIT_01.Sts_PVBad) TON(CS_Timer[67],?,?) XIC(CS_Timer[67].DN) ,XIC(AI_LIT_01.Sts_PVBad) TON(CS_Timer[70],?,?) XIC(CS_Timer[70].DN) ] [GRT(AI_LIT_01.Val,500) MOV(AI_LIT_01.Val,CS_REALParams[1]) ,LEQ(AI_LIT_01.Val,500) MOV(CS_REALParams[0],CS_REALParams[1]) ] MOV(CS_REALParams[1],CS_Result.FullDist) ,XIC(CS_Tank[LocalSampleTank].LeachOnly) ]XIC(Valve_XV_11.Sts_Closed)MOV(14,CS_Seq.ActiveStage);
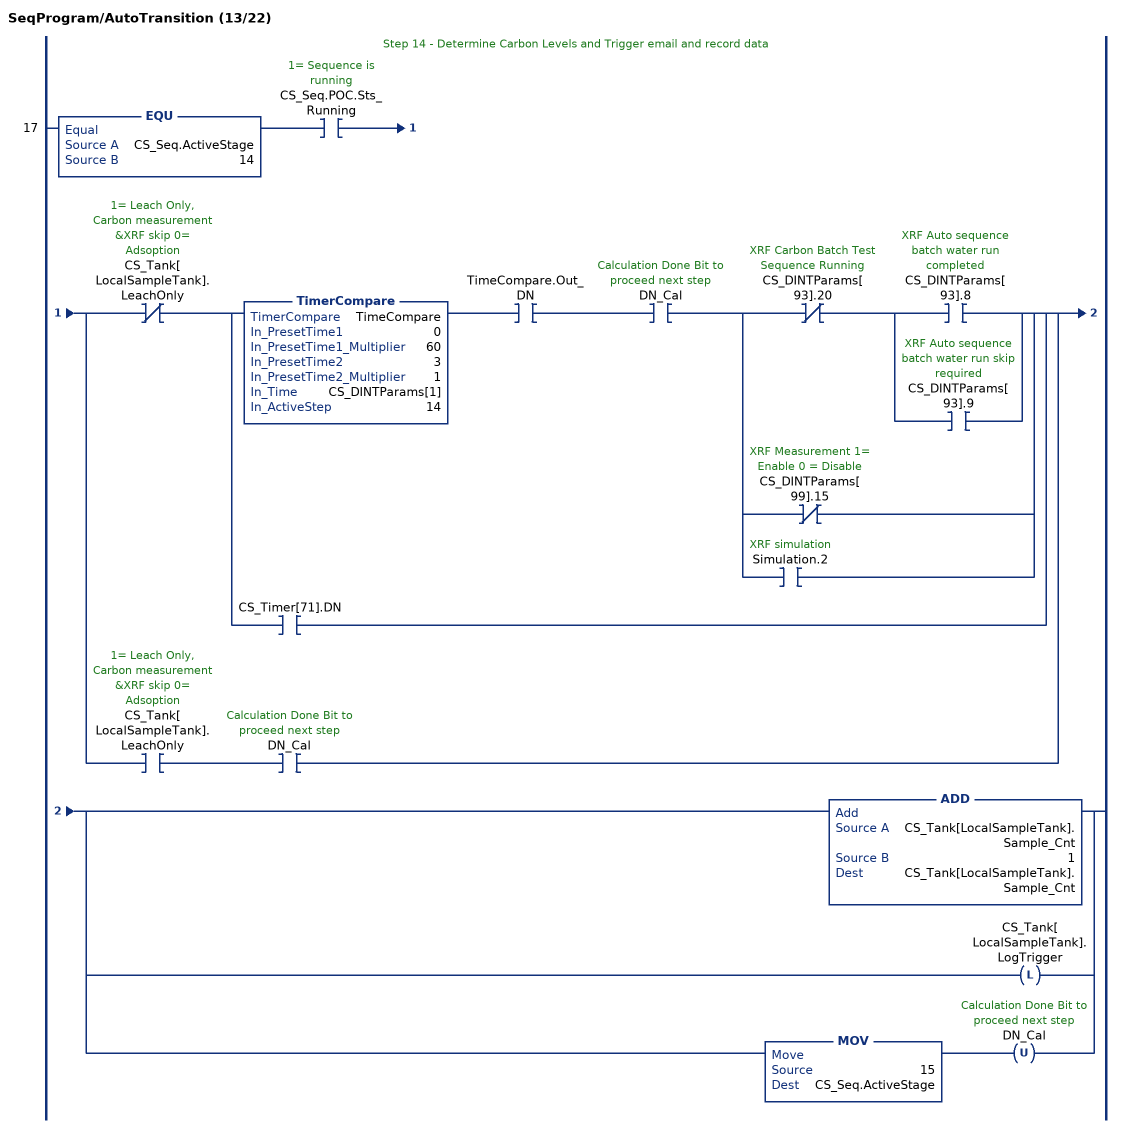
   // Step 14 - Determine Carbon Levels and Trigger email and record data
   17: EQU(CS_Seq.ActiveStage,14)XIC(CS_Seq.POC.Sts_Running)[XIO(CS_Tank[LocalSampleTank].LeachOnly) [TimerCompare(TimeCompare,0,60,3,1,CS_DINTParams[1],14) XIC(TimeCompare.Out_DN) XIC(DN_Cal) [XIO(CS_DINTParams[93].20) [XIC(CS_DINTParams[93].8) ,XIC(CS_DINTParams[93].9) ] ,XIO(CS_DINTParams[99].15) ,XIC(Simulation.2) ] ,XIC(CS_Timer[71].DN) ] ,XIC(CS_Tank[LocalSampleTank].LeachOnly) XIC(DN_Cal) ][ADD(CS_Tank[LocalSampleTank].Sample_Cnt,1,CS_Tank[LocalSampleTank].Sample_Cnt) ,OTL(CS_Tank[LocalSampleTank].LogTrigger) ,MOV(15,CS_Seq.ActiveStage) OTU(DN_Cal) ];
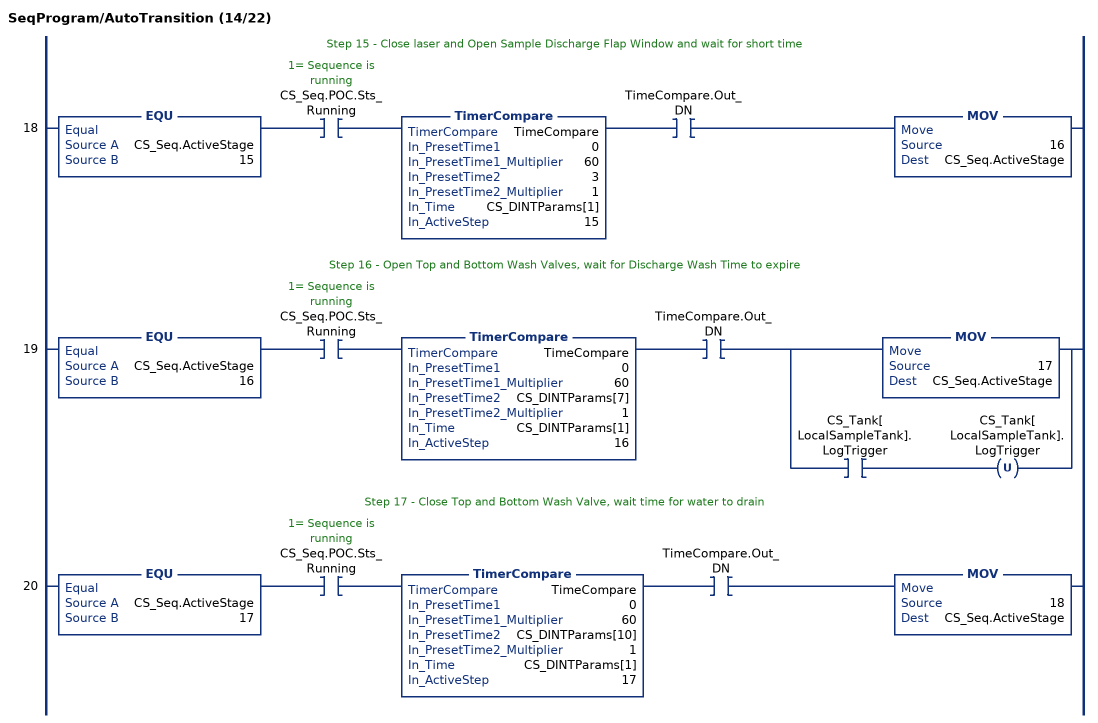
   // Step 15 - Close laser and Open Sample Discharge Flap Window and wait for short time
   18: EQU(CS_Seq.ActiveStage,15)XIC(CS_Seq.POC.Sts_Running)TimerCompare(TimeCompare,0,60,3,1,CS_DINTParams[1],15)XIC(TimeCompare.Out_DN)MOV(16,CS_Seq.ActiveStage);
   // Step 16 - Open Top and Bottom Wash Valves, wait for Discharge Wash Time to expire
   19: EQU(CS_Seq.ActiveStage,16)XIC(CS_Seq.POC.Sts_Running)TimerCompare(TimeCompare,0,60,CS_DINTParams[7],1,CS_DINTParams[1],16)XIC(TimeCompare.Out_DN)[MOV(17,CS_Seq.ActiveStage) ,XIC(CS_Tank[LocalSampleTank].LogTrigger) OTU(CS_Tank[LocalSampleTank].LogTrigger) ];
   // Step 17 - Close Top and Bottom Wash Valve, wait time for water to drain
   20: EQU(CS_Seq.ActiveStage,17)XIC(CS_Seq.POC.Sts_Running)TimerCompare(TimeCompare,0,60,CS_DINTParams[10],1,CS_DINTParams[1],17)XIC(TimeCompare.Out_DN)MOV(18,CS_Seq.ActiveStage);
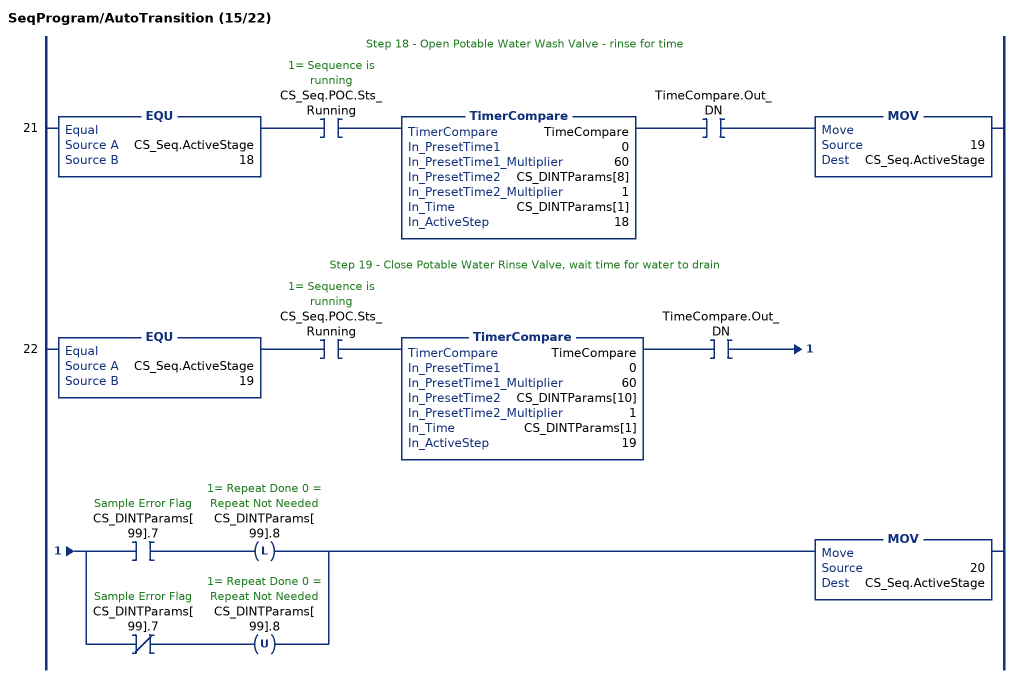
   // Step 18 - Open Potable Water Wash Valve - rinse for time
   21: EQU(CS_Seq.ActiveStage,18)XIC(CS_Seq.POC.Sts_Running)TimerCompare(TimeCompare,0,60,CS_DINTParams[8],1,CS_DINTParams[1],18)XIC(TimeCompare.Out_DN)MOV(19,CS_Seq.ActiveStage);
   // Step 19 - Close Potable Water Rinse Valve, wait time for water to drain
   22: EQU(CS_Seq.ActiveStage,19)XIC(CS_Seq.POC.Sts_Running)TimerCompare(TimeCompare,0,60,CS_DINTParams[10],1,CS_DINTParams[1],19)XIC(TimeCompare.Out_DN)[XIC(CS_DINTParams[99].7) OTL(CS_DINTParams[99].8) ,XIO(CS_DINTParams[99].7) OTU(CS_DINTParams[99].8) ]MOV(20,CS_Seq.ActiveStage);
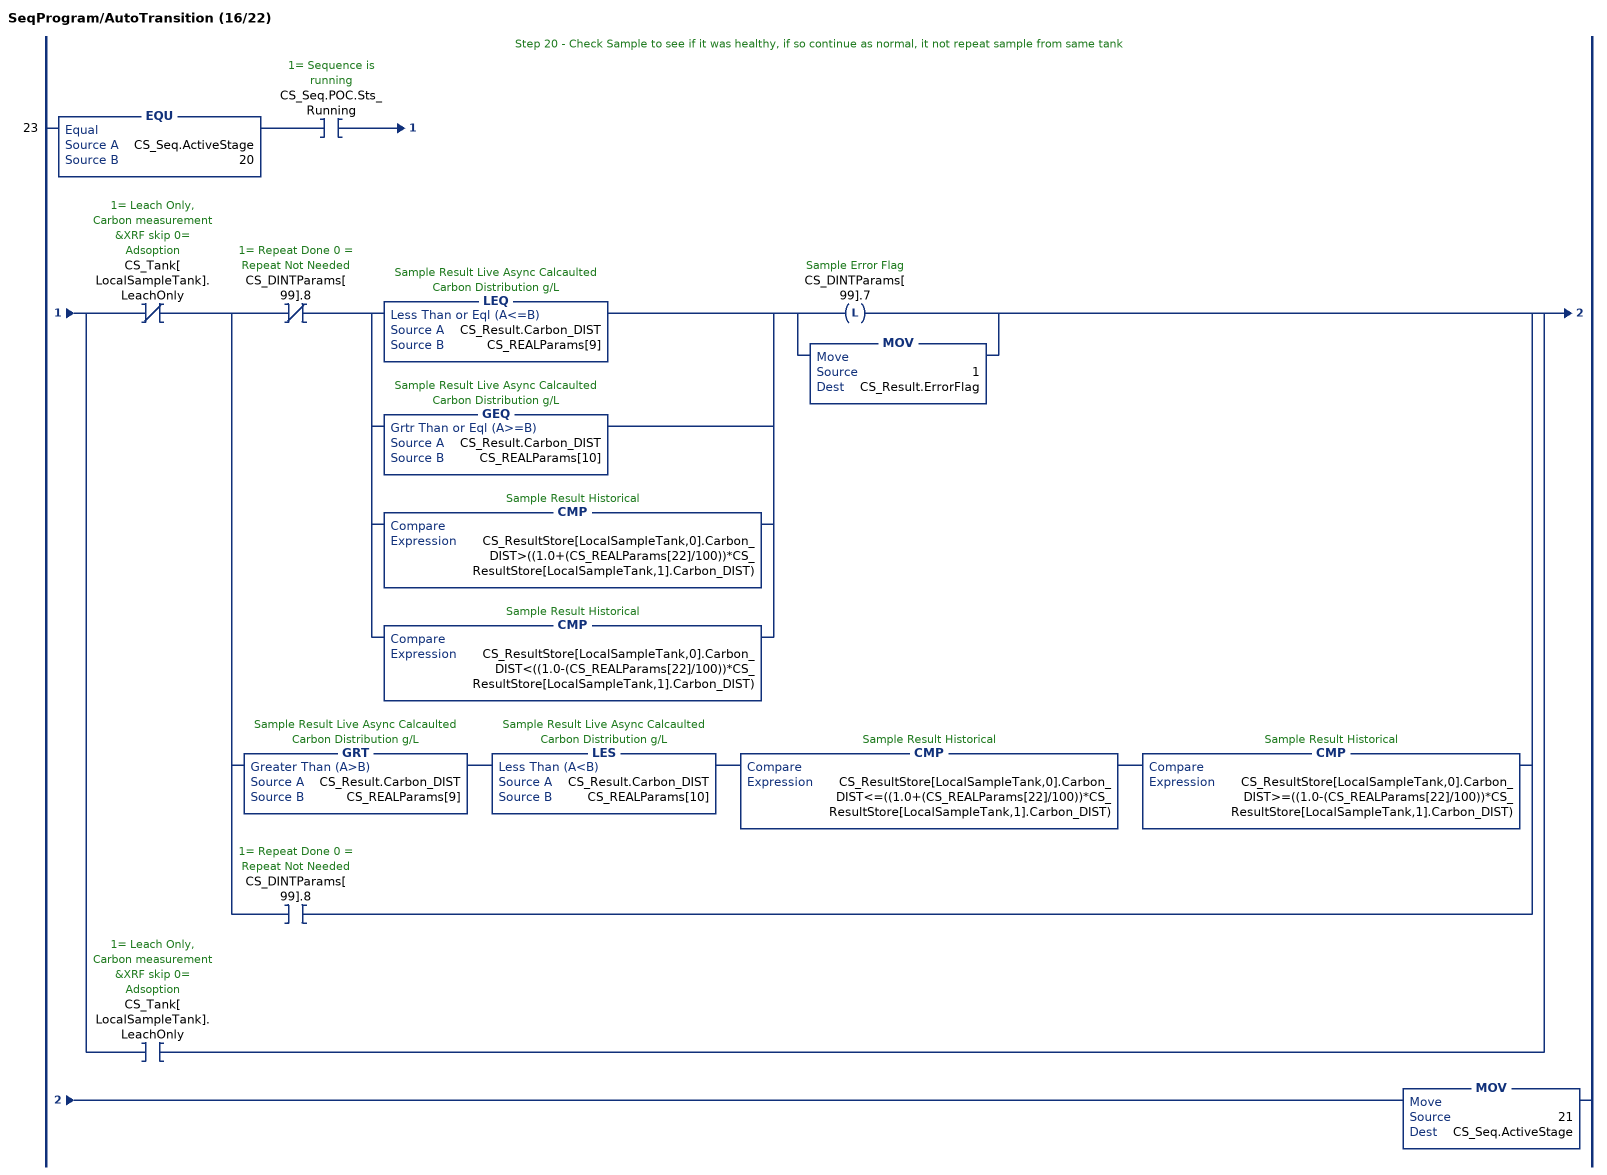
   // Step 20 - Check Sample to see if it was healthy, if so continue as normal, it not repeat sample from same tank
   23: EQU(CS_Seq.ActiveStage,20)XIC(CS_Seq.POC.Sts_Running)[XIO(CS_Tank[LocalSampleTank].LeachOnly) [XIO(CS_DINTParams[99].8) [LEQ(CS_Result.Carbon_DIST,CS_REALParams[9]) ,GEQ(CS_Result.Carbon_DIST,CS_REALParams[10]) ,CMP(CS_ResultStore[LocalSampleTank,0].Carbon_DIST>((1.0+(CS_REALParams[22]/100))*CS_ResultStore[LocalSampleTank,1].Carbon_DIST)) ,CMP(CS_ResultStore[LocalSampleTank,0].Carbon_DIST<((1.0-(CS_REALParams[22]/100))*CS_ResultStore[LocalSampleTank,1].Carbon_DIST)) ] [OTL(CS_DINTParams[99].7) ,MOV(1,CS_Result.ErrorFlag) ] ,GRT(CS_Result.Carbon_DIST,CS_REALParams[9]) LES(CS_Result.Carbon_DIST,CS_REALParams[10]) CMP(CS_ResultStore[LocalSampleTank,0].Carbon_DIST<=((1.0+(CS_REALParams[22]/100))*CS_ResultStore[LocalSampleTank,1].Carbon_DIST)) CMP(CS_ResultStore[LocalSampleTank,0].Carbon_DIST>=((1.0-(CS_REALParams[22]/100))*CS_ResultStore[LocalSampleTank,1].Carbon_DIST)) ,XIC(CS_DINTParams[99].8) ] ,XIC(CS_Tank[LocalSampleTank].LeachOnly) ]MOV(21,CS_Seq.ActiveStage);
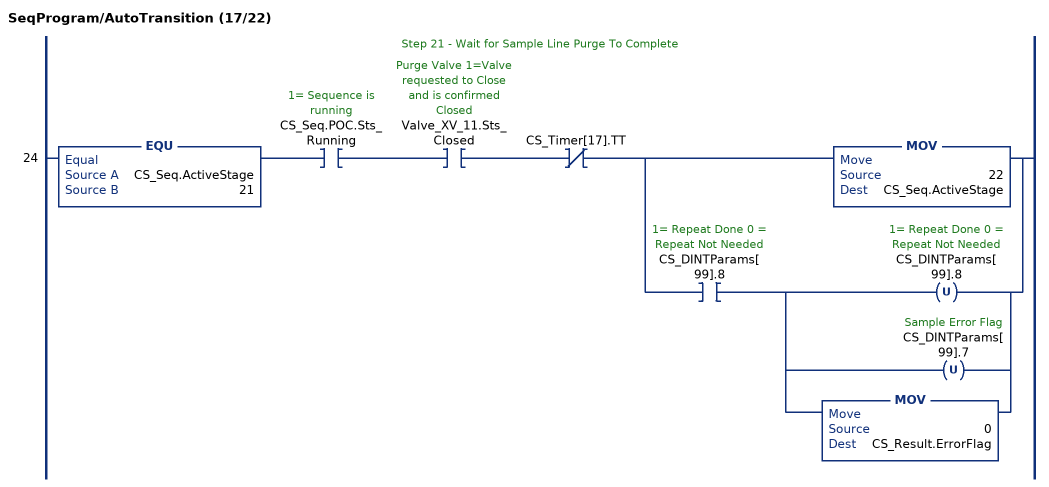
   // Step 21 - Wait for Sample Line Purge To Complete
   24: EQU(CS_Seq.ActiveStage,21)XIC(CS_Seq.POC.Sts_Running)XIC(Valve_XV_11.Sts_Closed)XIO(CS_Timer[17].TT)[MOV(22,CS_Seq.ActiveStage) ,XIC(CS_DINTParams[99].8) [OTU(CS_DINTParams[99].8) ,OTU(CS_DINTParams[99].7) ,MOV(0,CS_Result.ErrorFlag) ] ];
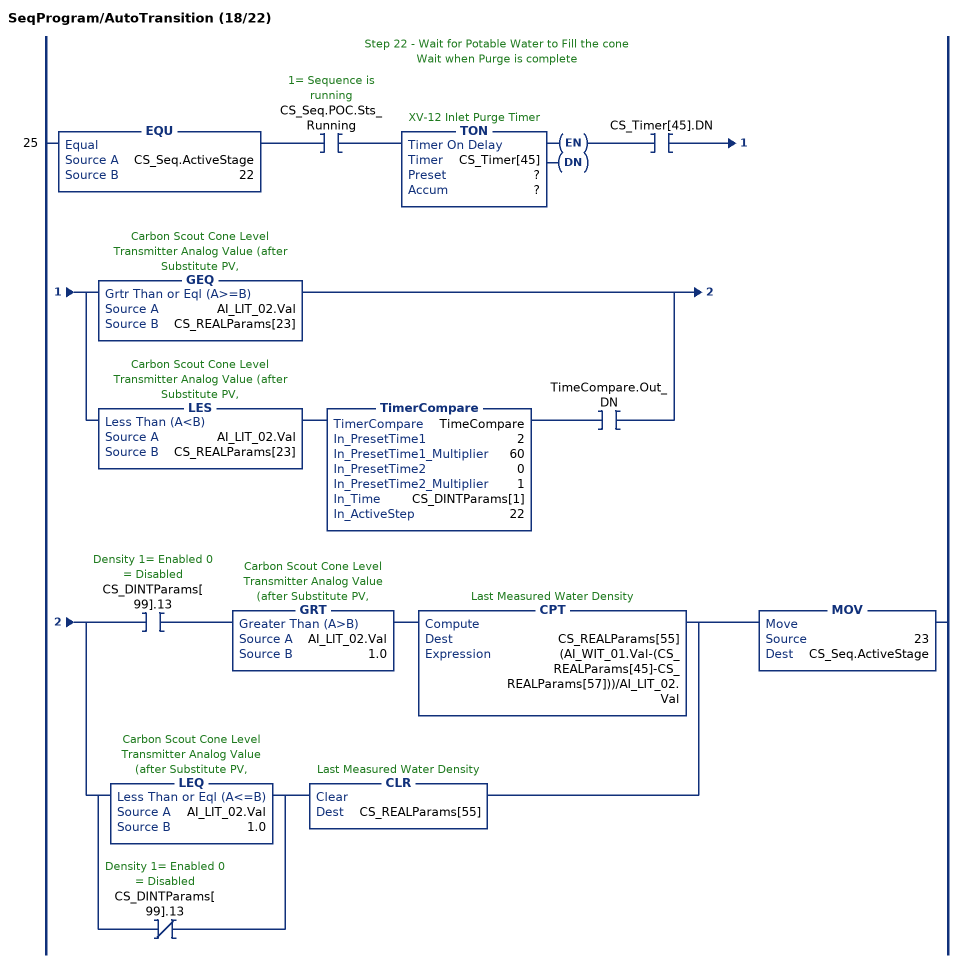
   // Step 22 - Wait for Potable Water to Fill the cone
   // Wait when Purge is complete
   25: EQU(CS_Seq.ActiveStage,22)XIC(CS_Seq.POC.Sts_Running)TON(CS_Timer[45],?,?)XIC(CS_Timer[45].DN)[GEQ(AI_LIT_02.Val,CS_REALParams[23]) ,LES(AI_LIT_02.Val,CS_REALParams[23]) TimerCompare(TimeCompare,2,60,0,1,CS_DINTParams[1],22) XIC(TimeCompare.Out_DN) ][XIC(CS_DINTParams[99].13) GRT(AI_LIT_02.Val,1.0) CPT(CS_REALParams[55],(AI_WIT_01.Val-(CS_REALParams[45]-CS_REALParams[57]))/AI_LIT_02.Val) ,[LEQ(AI_LIT_02.Val,1.0) ,XIO(CS_DINTParams[99].13) ] CLR(CS_REALParams[55]) ]MOV(23,CS_Seq.ActiveStage);
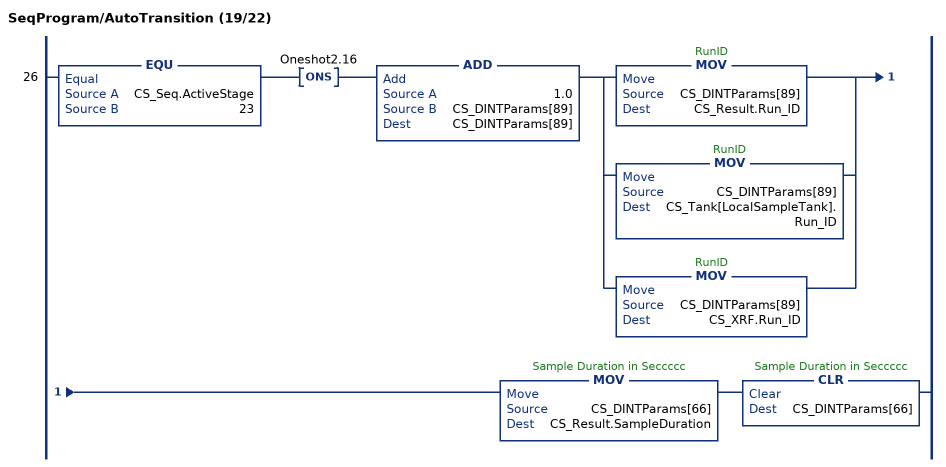
   26: EQU(CS_Seq.ActiveStage,23)ONS(Oneshot2.16)ADD(1.0,CS_DINTParams[89],CS_DINTParams[89])[MOV(CS_DINTParams[89],CS_Result.Run_ID) ,MOV(CS_DINTParams[89],CS_Tank[LocalSampleTank].Run_ID) ,MOV(CS_DINTParams[89],CS_XRF.Run_ID) ]MOV(CS_DINTParams[66],CS_Result.SampleDuration)CLR(CS_DINTParams[66]);
